// TIA Portal V17 export
// export: Created 2022-03-12T16:05:14.7765549Z, ExportSetting WithDefaults, DisplayName Totally Integrated Automation Portal, DisplayVersion V17, DisplayName TIA Portal Openness, DisplayVersion V17, DisplayName TIA Portal Version Control Interface, DisplayVersion V17, DisplayName STEP 7 Professional, DisplayVersion V17, DisplayName STEP 7 Safety, DisplayVersion V17, DisplayName WinCC Advanced / Unified PC, DisplayVersion V17
FUNCTION_BLOCK "UN_06_MiscFunctions"   // FB31626, LAD
TITLE = UN_06_MiscFunctions
{ S7_Optimized_Access := 'TRUE' }
AUTHOR : tech.team.motioncontrol@siemens.com
FAMILY : CPG
VERSION : 1.1
// Support: tech.team.motioncontrol@siemens.com
// stored: AutoNumber true, IsIECCheckEnabled false, IsRetainMemResEnabled false, MemoryReserve 100, SetENOAutomatically false, UDAEnableTagReadback false
   VAR
      instOEE_Calculation { ExternalAccessible := 'False'; ExternalVisible := 'False'; ExternalWritable := 'False'; S7_SetPoint := 'True'} : "CPG_OEE";   // FB used to calculate the real-time OEE value
      statOneShot_ProdConsumerCounter { ExternalAccessible := 'False'; ExternalVisible := 'False'; ExternalWritable := 'False'} : Bool;   // One Shot - products consumed counter
      statOneShot_ProdProcessedCounter { ExternalAccessible := 'False'; ExternalVisible := 'False'; ExternalWritable := 'False'} : Bool;   // One Shot - products processed counter
      statOneShot_ProdDefectiveCounter { ExternalAccessible := 'False'; ExternalVisible := 'False'; ExternalWritable := 'False'} : Bool;   // One Shot - products defective counter
   END_VAR
   VAR_TEMP
      tempReadClockRetVal : Int;
      tempProductionCounterTrigger : Bool;
   END_VAR
   VAR_TEMP   // added for the SCL form of the ladder/FBD networks
      _w1 : Bool;
   END_VAR
BEGIN

REGION Network 1: Update the PackTags Admin.PLC_Date_Time with current PLC time
   // 1) Update the "PackTags".Admin.PLC_Date_Time with the current PLC time.
   // 2) Update "HMI_Data".PLC_Date_Time.DATE_TIME with current PLC time so the HMI 
   // and PLC are time synchronized.
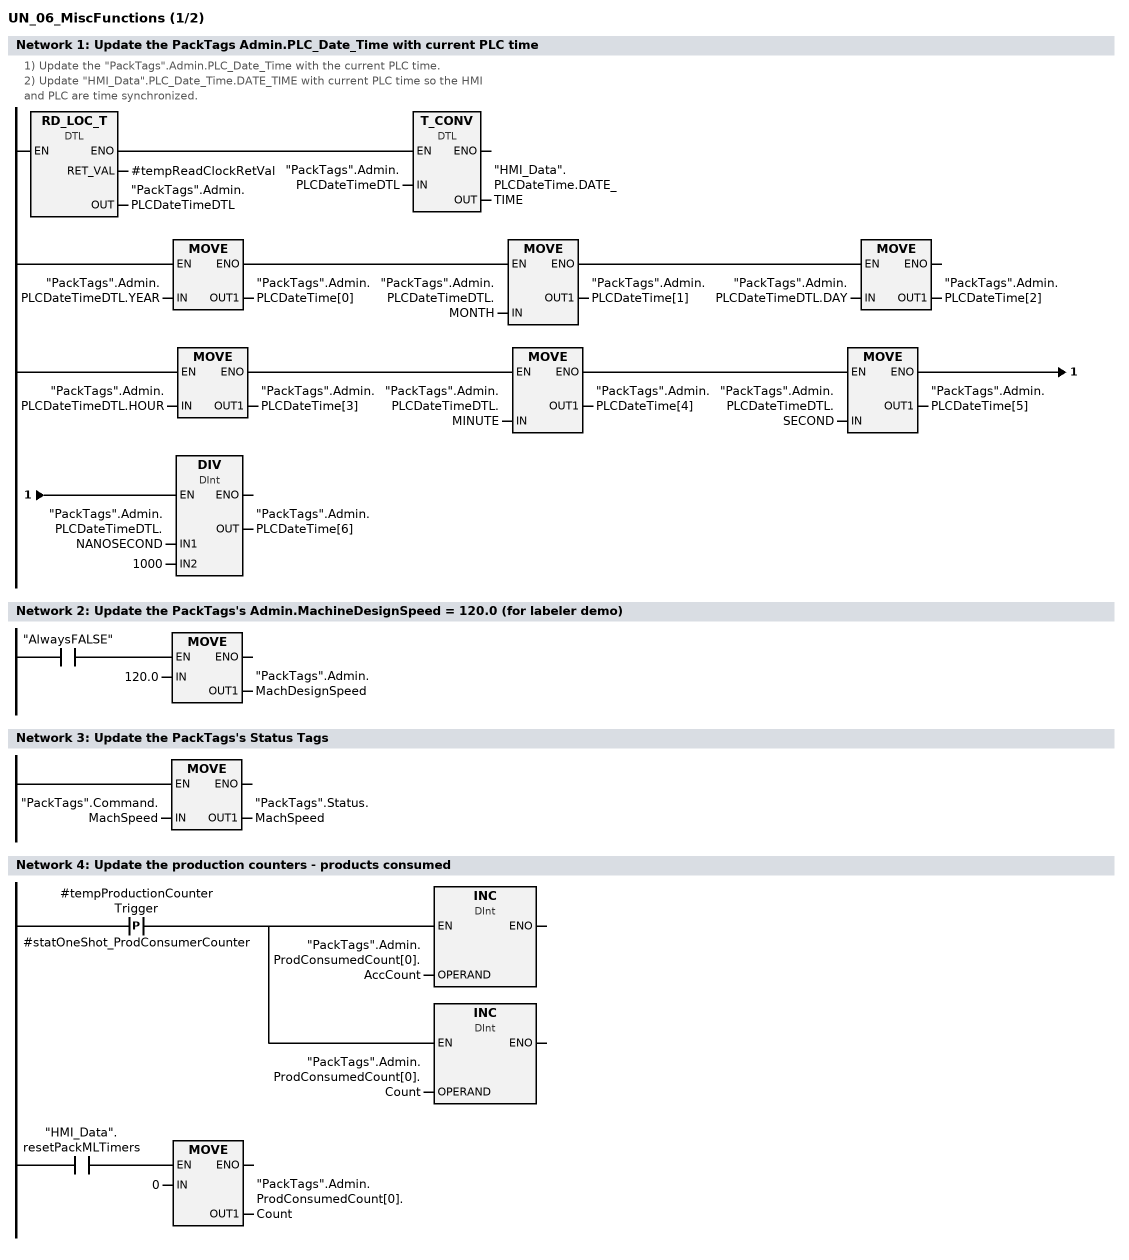
   RUNG wire#powerrail
      { S7_Templates := "date_type := DTL" } RD_LOC_T(RET_VAL => #tempReadClockRetVal, OUT => "PackTags".Admin.PLCDateTimeDTL)
      { S7_Templates := "[src_type := DTL, dest_type := Date_And_Time]" } T_CONV(IN := "PackTags".Admin.PLCDateTimeDTL, OUT => "HMI_Data".PLCDateTime.DATE_TIME)
   END_RUNG
   RUNG wire#powerrail
      Move(in := "PackTags".Admin.PLCDateTimeDTL.YEAR, out1 => "PackTags".Admin.PLCDateTime[0])
      Move(in := "PackTags".Admin.PLCDateTimeDTL.MONTH, out1 => "PackTags".Admin.PLCDateTime[1])
      Move(in := "PackTags".Admin.PLCDateTimeDTL.DAY, out1 => "PackTags".Admin.PLCDateTime[2])
   END_RUNG
   RUNG wire#powerrail
      Move(in := "PackTags".Admin.PLCDateTimeDTL.HOUR, out1 => "PackTags".Admin.PLCDateTime[3])
      Move(in := "PackTags".Admin.PLCDateTimeDTL.MINUTE, out1 => "PackTags".Admin.PLCDateTime[4])
      Move(in := "PackTags".Admin.PLCDateTimeDTL.SECOND, out1 => "PackTags".Admin.PLCDateTime[5])
      { S7_Templates := "SrcType := DInt" } Div(in1 := "PackTags".Admin.PLCDateTimeDTL.NANOSECOND, in2 := 1000, out => "PackTags".Admin.PLCDateTime[6])
   END_RUNG
   // the same network as SCL:
   #tempReadClockRetVal := RD_LOC_T(OUT => "PackTags".Admin.PLCDateTimeDTL, ENO => #_w1);
   IF #_w1 THEN
       T_CONV(IN := "PackTags".Admin.PLCDateTimeDTL, OUT => "HMI_Data".PLCDateTime.DATE_TIME);
   END_IF;
   "PackTags".Admin.PLCDateTime[0] := "PackTags".Admin.PLCDateTimeDTL.YEAR;
   "PackTags".Admin.PLCDateTime[1] := "PackTags".Admin.PLCDateTimeDTL.MONTH;
   "PackTags".Admin.PLCDateTime[2] := "PackTags".Admin.PLCDateTimeDTL.DAY;
   "PackTags".Admin.PLCDateTime[3] := "PackTags".Admin.PLCDateTimeDTL.HOUR;
   "PackTags".Admin.PLCDateTime[4] := "PackTags".Admin.PLCDateTimeDTL.MINUTE;
   "PackTags".Admin.PLCDateTime[5] := "PackTags".Admin.PLCDateTimeDTL.SECOND;
   "PackTags".Admin.PLCDateTime[6] := "PackTags".Admin.PLCDateTimeDTL.NANOSECOND / 1000;
END_REGION

REGION Network 2: Update the PackTags's Admin.MachineDesignSpeed = 120.0 (for labeler demo)
   RUNG wire#powerrail
      Contact( "AlwaysFALSE" )
      Move(in := 120.0, out1 => "PackTags".Admin.MachDesignSpeed)
   END_RUNG
   // the same network as SCL:
   IF "AlwaysFALSE" THEN "PackTags".Admin.MachDesignSpeed := 120.0; END_IF;
END_REGION

REGION Network 3: Update the PackTags's Status Tags
   RUNG wire#powerrail
      Move(in := "PackTags".Command.MachSpeed, out1 => "PackTags".Status.MachSpeed)
   END_RUNG
   // the same network as SCL:
   "PackTags".Status.MachSpeed := "PackTags".Command.MachSpeed;
END_REGION

REGION Network 4: Update the production counters - products consumed
   RUNG wire#powerrail
      P_Contact(operand := #tempProductionCounterTrigger, bit := #statOneShot_ProdConsumerCounter)
      wire#w1
      { S7_Templates := "DestType := DInt" } Inc( "PackTags".Admin.ProdConsumedCount[0].AccCount )
   END_RUNG
   RUNG wire#w1
      { S7_Templates := "DestType := DInt" } Inc( "PackTags".Admin.ProdConsumedCount[0].Count )
   END_RUNG
   RUNG wire#powerrail
      Contact( "HMI_Data".resetPackMLTimers )
      Move(in := 0, out1 => "PackTags".Admin.ProdConsumedCount[0].Count)
   END_RUNG
   // the same network as SCL:
   #_w1 := #tempProductionCounterTrigger AND NOT #statOneShot_ProdConsumerCounter;   // rising edge of #tempProductionCounterTrigger
   #statOneShot_ProdConsumerCounter := #tempProductionCounterTrigger;
   IF #_w1 THEN
       "PackTags".Admin.ProdConsumedCount[0].AccCount := "PackTags".Admin.ProdConsumedCount[0].AccCount + 1;
       "PackTags".Admin.ProdConsumedCount[0].Count := "PackTags".Admin.ProdConsumedCount[0].Count + 1;
   END_IF;
   IF "HMI_Data".resetPackMLTimers THEN "PackTags".Admin.ProdConsumedCount[0].Count := 0; END_IF;
END_REGION

REGION Network 5: Update the production counters - products processed
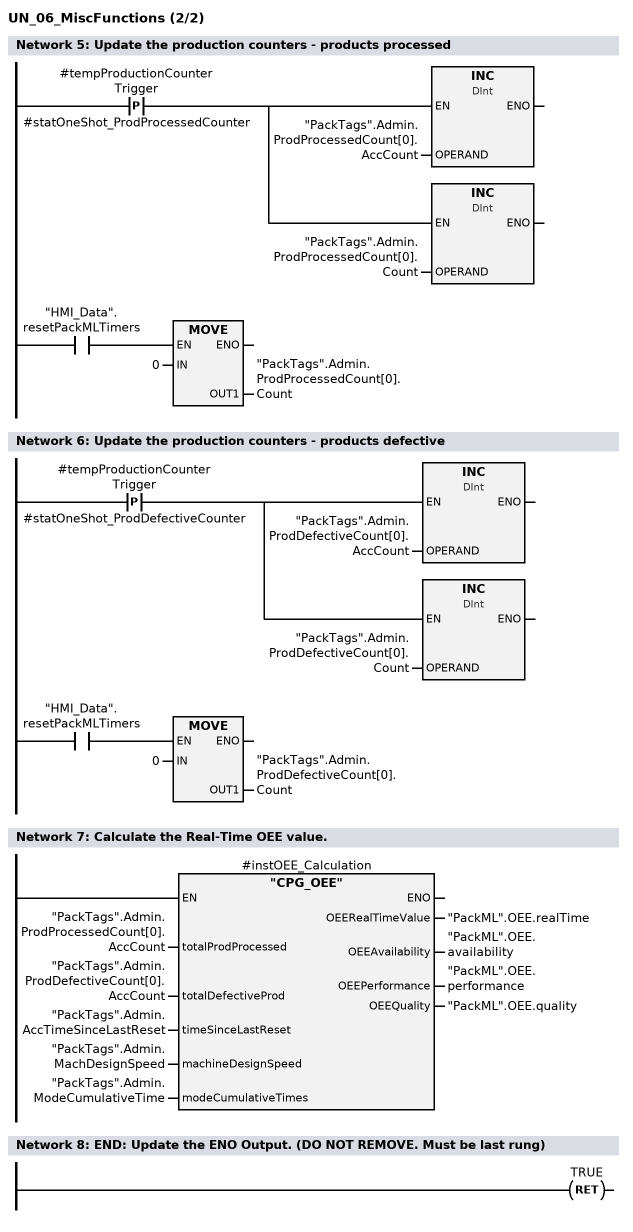
   RUNG wire#powerrail
      P_Contact(operand := #tempProductionCounterTrigger, bit := #statOneShot_ProdProcessedCounter)
      wire#w1
      { S7_Templates := "DestType := DInt" } Inc( "PackTags".Admin.ProdProcessedCount[0].AccCount )
   END_RUNG
   RUNG wire#w1
      { S7_Templates := "DestType := DInt" } Inc( "PackTags".Admin.ProdProcessedCount[0].Count )
   END_RUNG
   RUNG wire#powerrail
      Contact( "HMI_Data".resetPackMLTimers )
      Move(in := 0, out1 => "PackTags".Admin.ProdProcessedCount[0].Count)
   END_RUNG
   // the same network as SCL:
   #_w1 := #tempProductionCounterTrigger AND NOT #statOneShot_ProdProcessedCounter;   // rising edge of #tempProductionCounterTrigger
   #statOneShot_ProdProcessedCounter := #tempProductionCounterTrigger;
   IF #_w1 THEN
       "PackTags".Admin.ProdProcessedCount[0].AccCount := "PackTags".Admin.ProdProcessedCount[0].AccCount + 1;
       "PackTags".Admin.ProdProcessedCount[0].Count := "PackTags".Admin.ProdProcessedCount[0].Count + 1;
   END_IF;
   IF "HMI_Data".resetPackMLTimers THEN "PackTags".Admin.ProdProcessedCount[0].Count := 0; END_IF;
END_REGION

REGION Network 6: Update the production counters - products defective
   RUNG wire#powerrail
      P_Contact(operand := #tempProductionCounterTrigger, bit := #statOneShot_ProdDefectiveCounter)
      wire#w1
      { S7_Templates := "DestType := DInt" } Inc( "PackTags".Admin.ProdDefectiveCount[0].AccCount )
   END_RUNG
   RUNG wire#w1
      { S7_Templates := "DestType := DInt" } Inc( "PackTags".Admin.ProdDefectiveCount[0].Count )
   END_RUNG
   RUNG wire#powerrail
      Contact( "HMI_Data".resetPackMLTimers )
      Move(in := 0, out1 => "PackTags".Admin.ProdDefectiveCount[0].Count)
   END_RUNG
   // the same network as SCL:
   #_w1 := #tempProductionCounterTrigger AND NOT #statOneShot_ProdDefectiveCounter;   // rising edge of #tempProductionCounterTrigger
   #statOneShot_ProdDefectiveCounter := #tempProductionCounterTrigger;
   IF #_w1 THEN
       "PackTags".Admin.ProdDefectiveCount[0].AccCount := "PackTags".Admin.ProdDefectiveCount[0].AccCount + 1;
       "PackTags".Admin.ProdDefectiveCount[0].Count := "PackTags".Admin.ProdDefectiveCount[0].Count + 1;
   END_IF;
   IF "HMI_Data".resetPackMLTimers THEN "PackTags".Admin.ProdDefectiveCount[0].Count := 0; END_IF;
END_REGION

REGION Network 7: Calculate the Real-Time OEE value.
   RUNG wire#powerrail
      #instOEE_Calculation(totalProdProcessed := "PackTags".Admin.ProdProcessedCount[0].AccCount, totalDefectiveProd := "PackTags".Admin.ProdDefectiveCount[0].AccCount, timeSinceLastReset := "PackTags".Admin.AccTimeSinceLastReset, machineDesignSpeed := "PackTags".Admin.MachDesignSpeed, modeCumulativeTimes := "PackTags".Admin.ModeCumulativeTime, OEERealTimeValue => "PackML".OEE.realTime, OEEAvailability => "PackML".OEE.availability, OEEPerformance => "PackML".OEE.performance, OEEQuality => "PackML".OEE.quality)
   END_RUNG
   // the same network as SCL:
   #instOEE_Calculation(totalProdProcessed := "PackTags".Admin.ProdProcessedCount[0].AccCount,   // "CPG_OEE"
                        totalDefectiveProd := "PackTags".Admin.ProdDefectiveCount[0].AccCount,
                        timeSinceLastReset := "PackTags".Admin.AccTimeSinceLastReset,
                        machineDesignSpeed := "PackTags".Admin.MachDesignSpeed,
                        modeCumulativeTimes := "PackTags".Admin.ModeCumulativeTime,
                        OEERealTimeValue => "PackML".OEE.realTime,
                        OEEAvailability => "PackML".OEE.availability,
                        OEEPerformance => "PackML".OEE.performance,
                        OEEQuality => "PackML".OEE.quality);
END_REGION

REGION Network 8: END: Update the ENO Output. (DO NOT REMOVE. Must be last rung)
   RUNG wire#powerrail
      ReturnCoil( TRUE )
   END_RUNG
   // the same network as SCL:
   ENO := TRUE;
   RETURN;
END_REGION
END_FUNCTION_BLOCK
